Yaskawa INFORM job: TEST_TAKE_PICTURES.JBI

/JOB
//NAME TEST_TAKE_PICTURES
///FOLDERNAME TEST_JOBS
//POS
///NPOS 0,0,0,2,0,0
///USER 4
///TOOL 1
///POSTYPE USER
///RECTAN
///RCONF 1,0,0,0,0,0,0,0,0,0,0,0,0,0,0,0,0,0,0,0,0,0,0,0
P00001=-203.350,-49.507,11.578,0.0000,0.0000,0.0000
P00002=-198.450,-47.843,11.611,0.0000,0.0000,0.0000
//INST
///DATE 2022/11/08 12:30
///ATTR SC,RW
///GROUP1 RB1
NOP
CALL JOB:TAKE_PICTURES_OF_LINEAR_TRACE ARGFP001 ARGFP002 ARGF4 ARGF100000
END
